TYPE ST_St020_Interface :
STRUCT
	bEnableSequence,	// enable to main module
	
	bResponseChkIndex,
	bResponseIsEmptySlot,
	bResponseOpn	: BOOL;	// handshake response segment open
	iConfirmPosition	: INT;	// handshake confirm segment open @ x,y index
	
	Trolley			: TcaTrolley;
END_STRUCT
END_TYPE

(* stored: Version 1.1.0.1
   DUT ST_St020_Interface: Id {89d348a0-6b46-4a7a-8206-0f0c603c79cf} *)
